// TIA Portal V18 export
// export: Created 2025-12-01T17:50:33.8131352Z, ExportSetting None, DisplayName Totally Integrated Automation Portal, DisplayVersion V18 Update 5, DisplayName TIA Portal Openness, DisplayVersion V18 Update 5, DisplayName TIA Portal Teamcenter Gateway, DisplayVersion V18, DisplayName TIA Portal Version Control Interface, DisplayVersion V18, DisplayName STEP 7 Professional, DisplayVersion V18 Update 5, DisplayName STEP 7 Safety, DisplayVersion V18, DisplayName WinCC Professional, DisplayVersion V18 Update 5
DATA_BLOCK "ST10_WarningDB"   // DB1068
{ S7_Optimized_Access := 'FALSE' }
// stored: AutoNumber false
   VAR RETAIN
      Global : Struct   // Global Warning（通用警告）
         "1" : Struct
            PartLack1 : Bool;   // The main part1 lack
            PartLack2 : Bool;   // The part2 lack
            PartLack3 : Bool;   // The part3 lack
            PartLack4 : Bool;   // The part4 lack
            PartLack5 : Bool;   // The part5 lack
            PartLack6 : Bool;   // The part6 lack
            PartLack7 : Bool;   // The part7 lack
            PartLack8 : Bool;   // The part8 lack
         END_STRUCT;
         "2" : Array[0..15] of Bool;
         "3" : Struct
            PartNoProperPosition1 : Bool;   // The main part1 no proper position
            PartNoProperPosition2 : Bool;   // The part2 no proper position
            PartNoProperPosition3 : Bool;   // The part3 no proper position
            PartNoProperPosition4 : Bool;   // The part4 no proper position
            PartNoProperPosition5 : Bool;   // The part5 no proper position
            PartNoProperPosition6 : Bool;   // The part6 no proper position
            PartNoProperPosition7 : Bool;   // The part7 no proper position
            PartNoProperPosition8 : Bool;   // The part8 no proper position
         END_STRUCT;
         "4" : Array[0..15] of Bool;
         "5" : Struct
            ChangoverDataInvalide : Bool;   // The changover data invalide
            PartDateInvalide : Bool;   // The part date invalide
            StationInHPToStart : Bool;   // The station has to be at base pos to start
            lastStationPartNok : Bool;   // The last station part is Nok
         END_STRUCT;
         "6" : Array[0..15] of Bool;
         "7" : Array[0..15] of Bool;
         "8" : Array[0..15] of Bool;
         "9" : Array[0..15] of Bool;
         "10" : Array[0..15] of Bool;
      END_STRUCT;
      IndexTable : Array[1..2, 0..15] of Bool;   // Indextable Warning（转台警告）
      Serve : Array[1..2, 0..15] of Bool;   // Serve Warning（伺服警告）
      Servepress : Array[1..2, 0..15] of Bool;   // Serve press Warning（伺服压机警告）
      "3AxisServoInterpolation" : Array[1..2, 0..15] of Bool;   // Servo Motor Risk Money(3 axis)Warning （伺服电机3轴差补系统警告）
      LaserWelding : Array[1..2, 0..15] of Bool;   // Laser Welding Warning(激光焊接机警告)
      LaserMarking : Array[1..2, 0..15] of Bool;   // Laser Marking Warning(激光打标机警告)
      Printer : Array[1..2, 0..15] of Bool;   // Printer Warning(打印机警告)
      Marking : Array[1..2, 0..15] of Bool;   // Marking Warning(标识机警告)
      Labelling : Array[1..2, 0..15] of Bool;   // Labelling Warning（贴标机警告）
      Dispensing : Array[1..2, 0..15] of Bool;   // Dispensing Warning（点胶警告）
      GreasingSystem : Array[1..2, 0..15] of Bool;   // Greasing System Warning(注油系统警告）
      HotWindSystem : Array[1..2, 0..15] of Bool;   // Hot Wind System Warning(热风系统警告）
      HighFrequencyHeating : Array[1..2, 0..15] of Bool;   // High Frequency Heating Warning（高频加热警告）
      Degaussing : Array[1..2, 0..15] of Bool;   // Degaussing Warning（消磁警告）
      BowlFeeder : Array[1..2, 0..15] of Bool;   // Bowl Feeder Warning（振动盘警告）
      Riveter : Array[1..2, 0..15] of Bool;   // Riveter Warning（铆接机警告）
      HydraulicSystem : Array[1..2, 0..15] of Bool;   // Hydraulic System Warning（液压系统警告）
      Robot : Array[1..2, 0..15] of Bool;   // Robot Warning（机器人警告）
      Camera : Array[1..2, 0..15] of Bool;   // Camera Warning(影像警告)
      Scannner : Array[1..2, 0..15] of Bool;   // Scannner Warning(读码警告)
      MeasureSensor : Array[1..2, 0..15] of Bool;   // Measure Sensor Warning(测量传感器警告)
      Leakage : Array[1..2, 0..15] of Bool;   // Leakage Warning（泄露测试仪警告）
      TestPowerSupply : Array[1..2, 0..15] of Bool;   // Test Power Supply Warning (测试电源警告）
      HighVoltageTester : Array[1..2, 0..15] of Bool;   // High Voltage Test Warning(高压测试警告）
      EOLfinalInspection : Array[1..2, 0..15] of Bool;   // EOL final inspection Warning（EOL终检测试警告）
      Screw : Array[1..2, 0..15] of Bool;   // Screw Warning(电动螺丝刀警告)
      "3AxisScrewEncoder" : Array[1..2, 0..15] of Bool;   // Screw Encoder(3 axis)Warning(螺丝刀编码器警告）
      Heating : Array[1..2, 0..15] of Bool;   // Heating Warning（加热警告）
      PressurizedOilAirCylinder : Array[1..2, 0..15] of Bool;   // Pressurized Oil-Air Cylinder Warning(气液增力缸警告）
      Moby : Array[1..2, 0..15] of Bool;   // Moby Warning(Moby警告)
      IPC : Array[1..2, 0..15] of Bool;   // IPC Warning（服务器警告）
      ValveIsland : Array[1..2, 0..15] of Bool;   // Valve island Warning (阀岛警告）
      RFID : Array[1..2, 0..15] of Bool;   // RFID Warning（无线射频识别警告）
      RemoteIO : Array[1..2, 0..15] of Bool;   // Remote I/O Warning（远程I/O警告）
      DPSlaveStation : Array[1..2, 0..15] of Bool;   // DP Slave Station Warning（DP从站警告）
      MSCOMM : Array[1..2, 0..15] of Bool;   // MSCOMM Warning（串口通讯警告）
      Flowtester : Array[1..2, 0..15] of Bool;   // Flow tester Warning（流量测试仪错误）
      CurrentsTester : Array[1..2, 0..15] of Bool;   // Currents Tester Warning(电流测试仪)）
      VoltageTester : Array[1..2, 0..15] of Bool;   // Voltage Tester Warning(电压测试仪)
      InductanceTester : Array[1..2, 0..15] of Bool;   // Inductance Tester Warning(电感测试仪)
      ResistanceTester : Array[1..2, 0..15] of Bool;   // Resistance Tester Warning(电阻测试仪)
      LCRTester : Array[1..2, 0..15] of Bool;   // LCR Test Warning(LCR测试)
      PressureDisplacementMonitor : Array[1..2, 0..15] of Bool;   // Pressure Displacement Monitor Warning(压力位移监控仪)
      UltrasonicWelding : Array[1..2, 0..15] of Bool;   // Ultrasonic Welding Warning(超声波焊接)
      ElectricResistanceWelding : Array[1..2, 0..15] of Bool;   // Electric Resistance Welding Warning(电阻焊)
   END_VAR
BEGIN
END_DATA_BLOCK
